Fanuc KAREL source: kt00554.KL

-- PROVISIONAL review KL for V1013-1; original PC SHA256 341440d446c86cc9349df49e63cb79377aa99639916ad200fe36be8ca94419fb
-- Incomplete behavior may be omitted. Consult companion uncertainty JSON. Do not deploy.
PROGRAM KT00554
%NOLOCKGROUP
-- UNRESOLVED_DECL V1 type=000013
-- UNRESOLVED_DECL V2 type=000013
-- UNRESOLVED_DECL OUT type=000013
BEGIN
  -- UNRESOLVED_PC offsets 5-20; opcodes 2E,22,32,35
  -- UNRESOLVED_PC offsets 25-40; opcodes 2E,22,32,35
  -- UNRESOLVED_PC offsets 45-60; opcodes 2E,22,32,35
  -- UNRESOLVED_PC offsets 65-80; opcodes 2E,22,32,35
  -- UNRESOLVED_PC offsets 85-109; opcodes 49,49,92,4A
  -- UNRESOLVED_PC offsets 114-118; opcodes 7F
END KT00554
